// TIA Portal V15 export
// export: Created 2018-02-11T06:44:35.9001988Z, ExportSetting None, DisplayName Totally Integrated Automation Portal, DisplayVersion V15, DisplayName TIA Portal Openness, DisplayVersion V15, DisplayName TIA Portal Teamcenter Gateway, DisplayVersion V15, DisplayName SINAMICS Startdrive Advanced, DisplayVersion V15, DisplayName G110M, G120, G120C, G120D, G120P, DisplayVersion V15, DisplayName G130, G150, S120, S150, SINAMICS MV, DisplayVersion V15, DisplayName STEP 7 Professional, DisplayVersion V15, DisplayName WinCC Professional, DisplayVersion V15, DisplayName SIMATIC Visualization Architect, DisplayVersion V15
ORGANIZATION_BLOCK "Startup"   // OB100, LAD, Startup
TITLE = "Complete Restart"
{ S7_Optimized_Access := 'TRUE' }
// stored: SetENOAutomatically False
   VAR_INPUT
      LostRetentive : Bool;   // True if retentive data are lost
      LostRTC : Bool;   // True if date and time are lost
   END_VAR
BEGIN

REGION Network 1
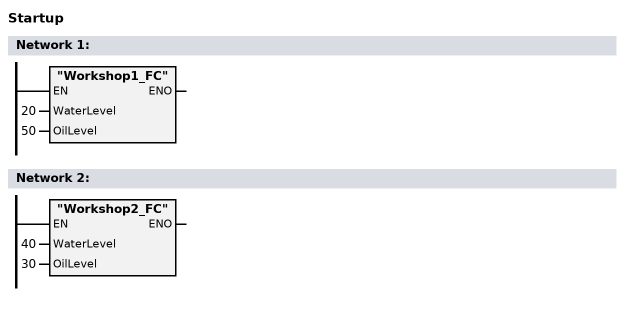
   RUNG wire#powerrail
      "Workshop1_FC"(WaterLevel := 20, OilLevel := 50)
   END_RUNG
   // the same network as SCL:
   "Workshop1_FC"(WaterLevel := 20, OilLevel := 50);
END_REGION

REGION Network 2
   RUNG wire#powerrail
      "Workshop2_FC"(WaterLevel := 40, OilLevel := 30)
   END_RUNG
   // the same network as SCL:
   "Workshop2_FC"(WaterLevel := 40, OilLevel := 30);
END_REGION
END_ORGANIZATION_BLOCK
